PROGRAM DatenRangieren
VAR	
	VersionsText: STRING := 'LAP 2010/1 Kompressoranlage V2.0';
END_VAR

VersionsInfo.Ver := MAXSTRING_TO_BYTEARR(VersionsText);

IF VersionsInfo.Befehle = 16#00 THEN	// lokale Ein- und Ausgänge verwenden
	SimDI.B1 := BitLesen(Plc_dSub.DI_LowByte,0);
	SimDI.B2 := BitLesen(Plc_dSub.DI_LowByte,1);
	SimDI.F1 := BitLesen(Plc_dSub.DI_LowByte,2);
	SimDI.S1 := BitLesen(Plc_dSub.DI_LowByte,3);
	SimDI.S2 := BitLesen(Plc_dSub.DI_LowByte,4);
		
	Plc_dSub.DQ_LowByte := AlleBitSetzen(	SimDa.P1,
											SimDa.P2,
											SimDa.Q1,
											SimDa.Q2,
											SimDa.Q3,	
											FALSE,	
											FALSE,										
											FALSE);	
ELSE	// Simulation (Digital Twin) verwenden
	SimDI.B1 := BitLesen(DigInput.DI[0],0);
	SimDI.B2 := BitLesen(DigInput.DI[0],1);
	SimDI.F1 := BitLesen(DigInput.DI[0],2);
	SimDI.S1 := BitLesen(DigInput.DI[0],3);
	SimDI.S2 := BitLesen(DigInput.DI[0],4);
	
	DigOutput.DA[0] := AlleBitSetzen(	SimDa.P1,
										SimDa.P2,
										SimDa.Q1,
										SimDa.Q2,
										SimDa.Q3,	
										FALSE,	
										FALSE,										
										FALSE);	
END_IF

END_PROGRAM

(* stored: Version 1.1.0.1, ProductVersion 3.1.4024.4
   POU DatenRangieren: Id {ad49a684-d9e6-4dba-bece-08745f191ac1}, SpecialFunc None *)
